(* CODESYS project Testment_Servo_Function_Test.export

Project tree, tasks and I/O mapping:
  Testment_Servo_Function_Test/
    program Servo_Testment_Main [ST]
    function block Testment_Message_Manager [ST]
*)

// Testment_Servo_Function_Test/Servo_Testment_Main
PROGRAM Servo_Testment_Main
VAR
	Set_Do: ARRAY [1..8] OF BOOL;
	Read_DI: ARRAY [1..12] OF BOOL;
	Read_DIA_Percentage :  ARRAY [0..7] OF REAL;
	Read_DIA_Raw :  ARRAY [0..7] OF UINT;
	
	// axis define
	FirstAxis : WORD := 1;
	LastAxis : WORD := 6;	// this value has been automaticlly asigned by global config reader
	//DI
	DI_Block : Digital_Input;
	
	//DO
	DO_Block : Digital_Output;
	
	//DIA
	smTime : TIME := T#250MS;
	DIA_Block : Digital_Input_Analog;
	
	
	// Testment functions
	Servo_Testment_State : INT := -1;
	Test_Process_Start_Restart, Error_State : BOOL;
	Message_Manager : Testment_Message_Manager;
	Show_Text : WSTRING;
	enb_axis : AuxAxis_PowerOn;
	read_axis : ARRAY [1..6] OF Arcalibrary.MCAT_ReadAxisMeasures;
	home_axis : ARRAY [1..6] OF Arcalibrary.MC_Home;
	re_j : INT;
	ts_i: INT;
	timer : ton;
	check_pos_err : REAL := 5;
	
	mov_axis : ARRAY [1..6] OF ArcaLibrary.MC_MoveAbsolute;
	FirstPos : REAL := 360;
	SecondPos : REAL := -360;
	CurrentPos : REAL;
	Vel : REAL := 180;
	Acc : REAL := 1900;
	Jerk : REAL := 9500;
	axis_mov_counter : INT;
	
	analog_cap ,analog_base : ARRAY [0..7] OF UINT;
	analog_difference : UINT := 12500; // 5v should be around 12900 ~ 13000
	set_override : ArcaLibrary.MC_GroupSetOverride;
	set_limit : ArcaLibrary.MCAT_AxisSetLimits;
	// analog control motor speed function
	analog_motor_state :INT := -1;
	debugButton : BOOL;
	speedLimit : REAL;
	analogFirPos : REAL := 380;
	analogSecPos : REAL := -380;
	analogVel : REAL := 18000;
	analogACC : REAL := 900000;
	analogJerk : REAL := 45000000;
	(* legacy ------
	forCounter: INT;
	//DI
	Read_6Ax_DI: Arcalibrary.ECAT_GetPdi_U32;
	DI_Raw : UDINT;
	new_DI_Value : UINT;
	
	//DO
	new_Do_Value, old_Do_Value : UINT;
	Write_6Ax_Do: Arcalibrary.ECAT_SetPdo_U32;
	------*)
	
	// servo elder program
	servo_elder_state :INT := -1;
	// elder_MoveType
	// 0 msans postion control all axis stop and turn in same time
	// 1 means speed control, two groups stop and turn in different times
	elder_MoveType : WORD := 1;
	elderVel : REAL := 18000;
	elderACC : REAL := 900000;
	elderJerk : REAL := 45000000;
	el_i : INT;
	speedFirGroup : ARRAY [0..5] OF ArcaLibrary.MC_MoveVelocity;
	speedSecGroup : ARRAY [0..5] OF ArcaLibrary.MC_MoveVelocity;
	elderTimer : ton;
	speedGroupSwitch : BOOL;
	speedSwitchTime : TIME := T#50MS;
	speedFirDir : ArcaLibrary.mc_Direction := mcPositiveDirection;
	speedSecDir : ArcaLibrary.mc_Direction := mcNegativeDirection;
	
	// 6 axis io test
	try: UINT;
	try2 : REAL;
	try3 : REAL := 3.9;
	read_0 : UINT;
	read_1 : UDINT;
	read_2 :ULINT;
	andValue : WORD;
	switch : BOOL;
	offsetValue : WORD := 147;
	TestAin_0: Arcalibrary.ECAT_GetPdi_U16;
	TestAin_1: Arcalibrary.ECAT_GetPdi_U32;
	TestAin_2: Arcalibrary.ECAT_GetPdi_U64;
	MaxmentOffset : UINT := 50;
	found_0, found_1, found_2, starter, maunl_next : BOOL;
	target_low : UINT := 12700;
	target_high : UINT := 13000;
	
	debugTimer : ton;
	FirstReachPos :  ARRAY [1..6] OF REAL := [0.6, -0.2, 0.606, -31.346, 178.434, 149.160];
	SecondReachPos :  ARRAY [1..6] OF REAL := [0.6, 0.2, 0.606, -31.346, 178.434, 149.160];
	Vell : REAL := 10;
	Accl : REAL := 10;
	Jerkl : REAL := 10;
	GrRelCorner :REAL := 0.5;
	MovErr : BOOL;
	//Movs : ARRAY [0..6] OF ArcaLibrary.MC_MoveLinearAbsolute;
	
	// error light control
	ErrLightControlState : INT;
	ErrLightTimer : Ton;
	ErrLightBlinkTime : TIME := T#200MS;
	ErrLightFinishTime : TIME := T#500MS;
	ErrLightCounterHigh : INT;
	ErrLightCounterLow : INT;
	ErrLight_i : INT;
	ErrLight_Switch : BOOL;
	// debug
	// --- because of homing bug (new servo need to home twice), get some function foe step 30
	homeErrOnce : BOOL;
	//---
	
	// debug
	manual_m01 : BOOL;
	manual_00 : BOOL;
	manual_20 : BOOL;
	manual_50 : BOOL;
	manual_jump_analog_check : BOOL;
	
	// debug para start---------------------------
	// read cfg message
	ReadCfg : ArcaLibrary.SYS_GetConfigInfo;
	Num_of_Axis:WORD;
	PowerState : ARRAY [0..5] OF ArcaLibrary.MCAT_ReadPowerStatus;
	AxisMeasure : ARRAY [0..5] OF ArcaLibrary.MCAT_ReadAxisMeasures;
	cfg_i : INT;
	
	//speed control test
	SC_Enb : BOOL; 
	SCMovTime : TIME := T#500MS;
	SCTimer : TON;
	SC_State : INT;
	SC_i,SC_y : INT;
	SpeedMovFir : ARRAY [0..5] OF ArcaLibrary.MC_MoveVelocity;
	SpeedMovSec : ARRAY [0..5] OF ArcaLibrary.MC_MoveVelocity;
	SCVel : REAL := 1800;
	SCACC : REAL := 9000;
	SCJerk : REAL := 45000;
	SCFirDir : ArcaLibrary.mc_Direction := mcPositiveDirection;
	SCSecDir : ArcaLibrary.mc_Direction := mcNegativeDirection;
	SCGroupSwitch : BOOL;
	
	// debug para end-----------------------------------
END_VAR

/////////////////////////////// instruction windows in chinsese  /////////////////////////////////////////

Message_Manager(state_in := Servo_Testment_State
	, start_restart_indicator => Test_Process_Start_Restart
	, Show_Message => Show_Text
	);
	
/////////////////////////////// instruction windows in chinsese  /////////////////////////////////////////

// if ethercat not ready then return
IF NOT ECatCfgok_GV THEN
	DI_Block (enable := FALSE);
	DO_Block (enable := FALSE);
	RETURN;
END_IF

IF Num_of_Axis_GV > 6 THEN
	Servo_Testment_State := -5;
END_IF
LastAxis := Num_of_Axis_GV;

DI_Block(enable := TRUE, DI_Array => Read_DI);
DO_Block(enable := TRUE, DO_Array := Set_Do);
DIA_Block(enable := TRUE, smoothTime := smTime
	, MaxRawInputValue := analog_cap
	, MinRawInputValue := analog_base
	, DIA_Raw => Read_DIA_Raw
	, DIA_Process => Read_DIA_Percentage
	);

enb_axis (enable := Servo_Testment_State > 9);
FOR re_j := 1 TO WORD_TO_INT(Num_of_Axis_GV) DO
	read_axis[re_j](axis := re_j - 1, enable :=  TRUE);
END_FOR

timer(in:= Servo_Testment_State = 30, pt := T#2S);

IF Servo_Testment_State <> -1 AND ((Read_DI[1] AND Read_DI[2]) OR manual_m01) THEN
	Servo_Testment_State := 0;
END_IF


set_limit(execute := debugButton, axis := 0, speedLimit := speedLimit); // useless

IF Servo_Testment_State < 130 THEN
	set_override(axesgroup := 0, enable := TRUE
	, velFactor := 1, accfactor := 1, jerkFactor := 1);
ELSE
	set_override(axesgroup := 0, enable := TRUE
	, velFactor := Read_DIA_Percentage[0]/100
	, accfactor := 1
	, jerkFactor := 1
	);
END_IF

IF Servo_Testment_State = 0 THEN	// reset
	//Set_Do[7]:= TRUE;
	//Set_Do[8]:= TRUE;
	homeErrOnce:= FALSE;
END_IF

CASE Servo_Testment_State OF
	-50: // analog cap and base difference too small
		// please connection and input voltage
		analog_cap[0];	// cap value
		analog_base[0];	// base vaule
	
	-45: // axis not mov to corrent pos
		ts_i; // error axis;
	-40: // if axis get err when moving
		ts_i; // error axis
	
	-35: // if some axis is not near 0 after homing
		ts_i; // error axis
		
	-33: // if some axis home err or time out
		ts_i;	// error axis
		
	-30: // if some axis home err
		home_axis[ts_i].ErrorID;	// homing err message
		
	-20: // if some axis can not enable
		enb_axis.Err_Message;	// enable err message
		
	-10: // if button is not commanding right inputs
		// plz check input button
		
	-5:	// config file contain more than 6 axis and exceed this program can handle
	
	-1:
		IF Read_DI[1] AND Read_DI[2] OR manual_m01 THEN
			Servo_Testment_State:= 0;
		ELSIF  Read_DI[1] OR Read_DI[2] THEN
			Servo_Testment_State := -10;	// if there is any input not receiving signal
		END_IF
		
	0:	// push second button to enable all axis
		IF Read_DI[3] AND Read_DI[4] AND Read_DI[5] AND Read_DI[6] OR manual_00 THEN
			Servo_Testment_State:= 10;
		ELSIF  Read_DI[3] OR Read_DI[4] OR Read_DI[5] OR Read_DI[6] THEN
			Servo_Testment_State := -10;	// if there is any input not receiving signal
		END_IF
	5:	// restart
		Servo_Testment_State := 10;
	10: // if 1~6 input is ok, waitting axis to enable
		IF enb_axis.Done THEN
			Servo_Testment_State := 20; // if enabled
		ELSIF enb_axis.Error THEN
			Servo_Testment_State := -20; // if some axis fail to enable
		END_IF
	20: // push third button to home axis
		FOR ts_i := WORD_TO_INT(FirstAxis) TO WORD_TO_INT(LastAxis) DO
			home_axis[ts_i](axis := ts_i - 1, execute := FALSE);	// reset blocks
		END_FOR
		IF Read_DI[7] AND Read_DI[8] AND Read_DI[9] OR homeErrOnce OR manual_20 THEN
			ts_i:= WORD_TO_INT(FirstAxis);
			Servo_Testment_State := 30;
		ELSIF Read_DI[7] OR Read_DI[8] OR Read_DI[9] THEN
			Servo_Testment_State := -10;	// if there is any input not receiving signal
		END_IF
	30: // start homing axis	// should not use I lkie in this case, is confilc with other state machine
		//Set_Do[7]:= TRUE;
		home_axis[ts_i](axis := ts_i - 1, execute := TRUE, position := 0, buffermode := mcAborting);
		IF home_axis[LastAxis].Done THEN	// all axis according to config file had homed
			FOR ts_i := WORD_TO_INT(FirstAxis) TO WORD_TO_INT(LastAxis) DO
				home_axis[ts_i](axis := ts_i - 1, execute := FALSE);
			END_FOR
			Servo_Testment_State := 40;
		ELSIF home_axis[ts_i].Done AND ts_i <= WORD_TO_INT(LastAxis) THEN // if current axis homing done
			timer(in:= FALSE);	// reset timer
			ts_i := ts_i + 1;
		ELSIF home_axis[ts_i].Error THEN	// if current axis get err
			Servo_Testment_State := -30;
		ELSIF timer.Q THEN	// if current axis not finish homing in certen time
			Servo_Testment_State := -33;
		END_IF
	40: // check if all axis are home
		ts_i := WORD_TO_INT(FirstAxis - 1);
		WHILE (ts_i < WORD_TO_INT(LastAxis)) AND Servo_Testment_State = 40 DO
			ts_i := ts_i + 1;
			IF read_axis[ts_i].Pos > check_pos_err OR read_axis[ts_i].Pos < -check_pos_err THEN // if current axis pos more than check_pos_err
				Servo_Testment_State := -35;
			END_IF
		END_WHILE
		IF Servo_Testment_State <> -35 THEN
			//Set_Do[8]:= TRUE;
			Servo_Testment_State := 50;
		END_IF
	50: // push fourth button to order motor turn
		FOR ts_i := WORD_TO_INT(FirstAxis) TO WORD_TO_INT(LastAxis) DO
			mov_axis[ts_i](axis := ts_i - 1, execute := FALSE);	// reset blocks
		END_FOR
		IF (Read_DI[10] AND Read_DI[11] AND Read_DI[12]) OR homeErrOnce OR manual_50 THEN
			Servo_Testment_State := 60;
		ELSIF Read_DI[10] OR Read_DI[11] OR Read_DI[12] THEN
			Servo_Testment_State := -10;	// if there is any input not receiving signal
		END_IF
	60:
		axis_mov_counter := 0;
		ts_i := WORD_TO_INT(FirstAxis - 1);
		WHILE ts_i < WORD_TO_INT(LastAxis) AND Servo_Testment_State = 60 DO
			ts_i := ts_i + 1;
			mov_axis[ts_i](axis := ts_i - 1, Execute := TRUE, Position := FirstPos
			, Velocity := vel, Acceleration := acc, Deceleration := Acc, jerk := jerk
			, Direction := mcShortestWay, BufferMode := mcAborting
			);
			IF mov_axis[ts_i].Done THEN
				axis_mov_counter := axis_mov_counter + 1;
			ELSIF  mov_axis[ts_i].Error THEN
				Servo_Testment_State := -40;	// axis err when moving
				IF NOT homeErrOnce THEN
					homeErrOnce := TRUE;
					Servo_Testment_State := 5;	// give secend chance
				END_IF
			END_IF
		END_WHILE
		IF axis_mov_counter >= WORD_TO_INT(LastAxis - (FirstAxis - 1)) AND Servo_Testment_State <> -40 THEN // if all axis mov done
			FOR ts_i := WORD_TO_INT(FirstAxis) TO WORD_TO_INT(LastAxis) DO
				mov_axis[ts_i](axis := ts_i - 1, execute := FALSE);	// reset blocks
			END_FOR
			Servo_Testment_State := 70;
		END_IF
	70: // check pos
		ts_i :=  WORD_TO_INT(FirstAxis - 1);
		WHILE ts_i < WORD_TO_INT(LastAxis) AND Servo_Testment_State = 70 DO
			ts_i := ts_i + 1;
			IF FirstPos - read_axis[ts_i].Pos < -check_pos_err OR FirstPos - read_axis[ts_i].Pos > check_pos_err THEN // if current axis pos more than check_pos_err
				Servo_Testment_State := -45;
			END_IF
		END_WHILE
		
		IF Servo_Testment_State <> -45 THEN
			Servo_Testment_State := 80;
		END_IF
		
	80: // motor start to turn
		axis_mov_counter := 0;
		ts_i := FirstAxis - 1;
		WHILE ts_i < WORD_TO_INT(LastAxis) AND Servo_Testment_State = 80 DO
			ts_i := ts_i + 1;
			mov_axis[ts_i](axis := ts_i - 1, Execute := TRUE, Position := SecondPos
			, Velocity := vel, Acceleration := acc, Deceleration := Acc, jerk := jerk
			, Direction := mcShortestWay, BufferMode := mcAborting
			);
			IF mov_axis[ts_i].Done THEN
				axis_mov_counter := axis_mov_counter + 1;
			ELSIF  mov_axis[ts_i].Error THEN
				Servo_Testment_State := -40;	// axis err when moving
			END_IF
		END_WHILE
		IF axis_mov_counter >= LastAxis - (FirstAxis - 1) AND Servo_Testment_State <> -40 THEN // if all axis mov done
			Servo_Testment_State := 90;
		END_IF
		
	90: // check pos
		ts_i := FirstAxis - 1;
		WHILE ts_i < WORD_TO_INT(LastAxis) AND Servo_Testment_State = 90 DO
			ts_i := ts_i + 1;
			IF SecondPos - read_axis[ts_i].Pos < -check_pos_err OR SecondPos - read_axis[ts_i].Pos > check_pos_err THEN // if current axis pos more than check_pos_err
				Servo_Testment_State := -45;
			END_IF
		END_WHILE
		IF Servo_Testment_State <> -45 THEN
			FOR ts_i := WORD_TO_INT(FirstAxis) TO WORD_TO_INT(LastAxis) DO
				mov_axis[ts_i](axis := ts_i - 1, execute := FALSE);	// reset blocks
			END_FOR
			Servo_Testment_State := 100;
		END_IF
		
	100: // set analog input base value, click second button to remember
		analog_base[0] := Read_DIA_Raw[0];
		IF Read_DI[3] AND Read_DI[4] AND Read_DI[5] AND Read_DI[6] OR manual_jump_analog_check THEN
			Servo_Testment_State:= 110;
		ELSIF  Read_DI[3] OR Read_DI[4] OR Read_DI[5] OR Read_DI[6] THEN
			Servo_Testment_State := -10;	// if there is any input not receiving signal
		END_IF
		
	110: // set analog input cap value, click third button to remember
		analog_cap[0] := Read_DIA_Raw[0];
		IF Read_DI[7] AND Read_DI[8] AND Read_DI[9] OR manual_jump_analog_check THEN
			Servo_Testment_State := 120;
		ELSIF Read_DI[7] OR Read_DI[8] OR Read_DI[9] THEN
			Servo_Testment_State := -10;	// if there is any input not receiving signal
		END_IF
		
	120: // check difference between cap and base
		IF (analog_cap[0] - analog_base[0] > analog_difference) OR manual_jump_analog_check THEN
			Servo_Testment_State := 130;
		ELSE
			Servo_Testment_State := -50;
		END_IF
	130:
		
	//100: // procedure done
		
END_CASE

(*IF Servo_Testment_State < 130 THEN
	analog_motor_state := -1;
END_IF

(*************
original Servo_Testment_State > 130 is designed for analog control axis speed
currently this state is use for servo elder testment
*******************)
CASE analog_motor_state	OF

	-1:
		//analog_motor_state := 0;
	0:
		FOR i := 1 TO WORD_TO_INT(Num_of_Axis_GV) DO	// should not use I here because this I is conflic with test state
			mov_axis[i](axis := i - 1, execute := FALSE);	// reset blocks
		END_FOR
		analog_motor_state := 10;
		debugTimer(in:= FALSE);
		(*
	10:
		mov_axis[1](axis := 0, Execute := TRUE, Position := 0);
		mov_axis[2](axis := 1, Execute := TRUE, Position := 0);
		mov_axis[3](axis := 2, Execute := TRUE, Position := 0);
		mov_axis[4](axis := 3, Execute := TRUE, Position := 0);
		mov_axis[5](axis := 4, Execute := TRUE, Position := 0);
		mov_axis[6](axis := 5, Execute := TRUE, Position := 0);
		debugTimer (in:= TRUE, pt := T#5S);
		IF debugTimer.Q THEN
			debugTimer(in:= FALSE);
			
			FOR i := 1 TO WORD_TO_INT(Num_of_Axis_GV) DO
				mov_axis[i](axis := i - 1, execute := FALSE);	// reset blocks
			END_FOR
			analog_motor_state := 20;
			
			Movs[0](axesgroup := 0, Execute := FALSE);
			
			Movs[1](axesgroup := 0, Execute := FALSE);
		END_IF
		
	20:
		Movs[0](axesgroup := 0, Execute := TRUE, Position := ADR(FirstReachPos)
			, Velocity := vell, Acceleration := accl, Deceleration := Accl, jerk := jerkl
			, coordsystem := mcMcs, BufferMode := mcAborting
			, TransitionMode := tmNone, TransitionParameter:=ADR(GrRelCorner)
			, Error => MovErr);
		IF Movs[0].Done THEN
			Movs[0](axesgroup := 0, Execute := FALSE);
			analog_motor_state := 30;
		END_IF
	30:
		Movs[1](axesgroup := 0, Execute := TRUE, Position := ADR(SecondReachPos)
			, Velocity := vell, Acceleration := accl, Deceleration := Accl, jerk := jerkl
			, coordsystem := mcMcs, BufferMode := mcAborting
			, TransitionMode := tmNone, TransitionParameter:=ADR(GrRelCorner)
			, Error => MovErr);
		IF Movs[1].Done THEN
			Movs[1](axesgroup := 0, Execute := FALSE);
			analog_motor_state := 20;
		END_IF
	*)
END_CASE*)

IF Servo_Testment_State < 130 THEN
	servo_elder_state := -1;
END_IF
CASE servo_elder_state OF
	-1:
		IF elder_MoveType = 0 THEN	// if control in abs 
			servo_elder_state := 0;
		ELSIF elder_MoveType = 1 THEN	// if control in vel
			servo_elder_state := 30;
		END_IF
	0:
		FOR el_i := 1 TO WORD_TO_INT(Num_of_Axis_GV) DO
			mov_axis[el_i](axis := el_i - 1, execute := FALSE);	// reset blocks
		END_FOR
		
		servo_elder_state := 10;
	10:
		axis_mov_counter := 0;
		el_i := 0;
		WHILE el_i < WORD_TO_INT(LastAxis - (FirstAxis - 1)) AND Servo_Testment_State <> -40 DO
			el_i := el_i + 1;
			mov_axis[el_i](axis := el_i - 1, Execute := TRUE, Position := analogFirPos
				, velocity := elderVel, Acceleration := elderACC, Deceleration := elderACC, Jerk := elderJerk
				, Direction := mcShortestWay, BufferMode := mcAborting
			);
			IF mov_axis[el_i].Done THEN
				axis_mov_counter := axis_mov_counter + 1;
			ELSIF  mov_axis[el_i].Error THEN
				Servo_Testment_State := -40;	// axis err when moving
			END_IF
		END_WHILE
		IF axis_mov_counter >= 6 AND Servo_Testment_State <> -40 THEN // if all axis mov done
			FOR el_i := WORD_TO_INT(FirstAxis) TO WORD_TO_INT(LastAxis) DO
				mov_axis[el_i](axis := el_i - 1, execute := FALSE);	// reset blocks
			END_FOR
			servo_elder_state := 20;
		END_IF
	20:
		axis_mov_counter := 0;
		el_i := 0;
		WHILE el_i < WORD_TO_INT(LastAxis - (FirstAxis - 1)) AND Servo_Testment_State <> -40 DO
			el_i := el_i + 1;
			mov_axis[el_i](axis := el_i - 1, Execute := TRUE, Position := analogSecPos
				, velocity := elderVel, Acceleration := elderACC, Deceleration := elderACC, Jerk := elderJerk
				, Direction := mcShortestWay, BufferMode := mcAborting
			);
			IF mov_axis[el_i].Done THEN
				axis_mov_counter := axis_mov_counter + 1;
			ELSIF  mov_axis[el_i].Error THEN
				Servo_Testment_State := -40;	// axis err when moving
			END_IF
		END_WHILE
		IF axis_mov_counter >= 6 AND Servo_Testment_State <> -40 THEN // if all axis mov done
			FOR el_i := WORD_TO_INT(FirstAxis) TO WORD_TO_INT(LastAxis) DO
				mov_axis[el_i](axis := el_i - 1, execute := FALSE);	// reset blocks
			END_FOR
			servo_elder_state := 10;
		END_IF
	30:
		FOR el_i := 0 TO 5 DO
			speedFirGroup[el_i](axis := el_i,execute := FALSE);
			speedSecGroup[el_i](axis := el_i,execute := FALSE);
		END_FOR
		elderTimer(in := FALSE);
		speedGroupSwitch := FALSE;
		servo_elder_state := 40;
	40:
		elderTimer(in := TRUE, pt := speedSwitchTime);
		IF elderTimer.Q THEN	// if time reached
			IF NOT speedGroupSwitch THEN	//decide which motor group is time to switch dir
				speedGroupSwitch := TRUE;
				IF speedFirDir = mcPositiveDirection THEN	// if first group is moving positivily
					speedFirDir := mcNegativeDirection;	// then switch to negative
				ELSE
					speedFirDir := mcPositiveDirection;
				END_IF
			ELSE
				speedGroupSwitch := FALSE;
				IF speedSecDir = mcPositiveDirection THEN
					speedSecDir := mcNegativeDirection;
				ELSE
					speedSecDir := mcPositiveDirection;
				END_IF
			END_IF
		END_IF
		FOR el_i := 0 TO 5 BY 2 DO
			speedFirGroup[el_i](axis := el_i,execute := NOT (elderTimer.Q AND speedGroupSwitch)	// only switch off when timer is alarted and first group direction is switched
				, velocity := elderVel, Acceleration := elderACC, Deceleration := elderACC, Jerk := elderJerk
				, Direction := speedFirDir, Buffermode := mcAborting);
			IF  speedFirGroup[el_i].Error THEN
				Servo_Testment_State := -40;	// axis err when moving
			END_IF
		END_FOR
		FOR el_i := 1 TO 5 BY 2 DO
			speedFirGroup[el_i](axis := el_i,execute := NOT (elderTimer.Q AND NOT speedGroupSwitch)	// only switch off when timer is alarted and second group direction is switched
				, velocity := elderVel, Acceleration := elderACC, Deceleration := elderACC, Jerk := elderJerk
				, Direction := speedSecDir, Buffermode := mcAborting);
			IF  speedFirGroup[el_i].Error THEN
				Servo_Testment_State := -40;	// axis err when moving
			END_IF
		END_FOR
		
		IF elderTimer.Q THEN	// if time reached
			elderTimer(in := FALSE);	// switch off timer
		END_IF
END_CASE

IF Servo_Testment_State > -1 THEN
	errlightcontrolstate := 0;
END_IF
CASE errlightcontrolstate OF
	0:
		Set_Do[7]:= TRUE;
		Set_Do[8]:= TRUE;
		IF Servo_Testment_State < 0 THEN
			Set_Do[7]:= FALSE;
			Set_Do[8]:= FALSE;
			ErrLightCounterHigh := (ABS(Servo_Testment_State) / 10) MOD 10;
			ErrLightCounterLow := ABS(Servo_Testment_State) MOD 10;
			ErrLightTimer(in := FALSE);
			ErrLight_i := 0;
			ErrLight_Switch := FALSE;
			IF ErrLightCounterHigh > 0 THEN
				errlightcontrolstate := 10;	// if there have higer num next state
			ELSE
				errlightcontrolstate := 20;	// go to low num directily
			END_IF
		END_IF
	10:	// blink higher number
		Set_Do[7]:= ErrLight_Switch;
		ErrLightTimer(in := TRUE , pt:= ErrLightBlinkTime);
		IF ErrLightTimer.Q THEN
			IF ErrLight_Switch THEN
				ErrLight_Switch := FALSE;
			ELSE
				ErrLight_Switch := TRUE;
			END_IF
			ErrLightTimer (in := FALSE);
			ErrLight_i := ErrLight_i + 1;
		END_IF
		IF ErrLight_i >= (ErrLightCounterHigh * 2) THEN
			ErrLightTimer(in := FALSE);
			ErrLight_i := 0;
			ErrLight_Switch := FALSE;
			IF ErrLightCounterLow > 0 THEN
				errlightcontrolstate := 20;	// if have lower num
			ELSE
				errlightcontrolstate := 30;	// go wating time
			END_IF
		END_IF
	20:// blink lower number
		Set_Do[8]:= ErrLight_Switch;
		ErrLightTimer(in := TRUE , pt:= ErrLightBlinkTime);
		IF ErrLightTimer.Q THEN
			IF ErrLight_Switch THEN
				ErrLight_Switch := FALSE;
			ELSE
				ErrLight_Switch := TRUE;
			END_IF
			ErrLightTimer (in := FALSE);
			ErrLight_i := ErrLight_i + 1;
		END_IF
		IF ErrLight_i >= (ErrLightCounterLow * 2) THEN
			ErrLightTimer(in := FALSE);
			ErrLight_i := 0;
			ErrLight_Switch := FALSE;
			errlightcontrolstate := 30;	// next state
		END_IF
	30:
		ErrLightTimer(in := TRUE, pt := ErrLightFinishTime);
		IF ErrLightTimer.Q THEN
			errlightcontrolstate := 0;
		END_IF
END_CASE

(* legacy ------
// read di
Read_6Ax_DI(Enable:=Num_of_axis_GV > 0, Offset:=143, Value=>DI_Raw);
new_DI_Value := UDINT_TO_UINT(DI_Raw);	// need convert to UINT otherwise it contain much more unwanted bits, it's not necessary but just keep this line to remember
// judge which bit is true
FOR forCounter := 1 TO UINT_TO_INT(SIZEOF(Read_DI)) DO // loop all bool value
	Read_DI[forCounter] := UINT_TO_BOOL(new_DI_Value AND SHL(1, forCounter - 1));
END_FOR

// write do
new_Do_Value:= 0;	// initialize 

(*	useless too complicated, no need to do the real calculation
FOR forCounter := 0 TO UINT_TO_INT(SIZEOF(SetDo)) DO // loop all bool value
	IF SetDo[forCounter] THEN	// if out put is true
		squareValue := 1;	// first value is 1, 2^0=1
		IF forCounter <> 0 THEN // if is not first value
			FOR squareCounter := 1 TO forCounter DO	// calculate dec value
				squareValue := squareValue * 2;
			END_FOR
		END_IF
		DoValue := DoValue + INT_TO_UINT(squareValue);
	END_IF
END_FOR
*)
// shift mamary according to bool
FOR forCounter := 1 TO UINT_TO_INT(SIZEOF(Set_Do)) DO // loop all bool value
	IF Set_Do[forCounter] THEN	// if out put is true
		new_Do_Value := new_Do_Value + SHL(1, forCounter - 1);
	END_IF
END_FOR

IF new_Do_Value <> old_Do_Value THEN
	old_Do_Value := new_Do_Value;
END_IF
Write_6Ax_Do(Enable:=Num_of_axis_GV > 0, Offset:=143, Value:=old_Do_Value);	// write DO
---------*)
// debug
IF NOT starter THEN
	starter := TRUE;
	found_0 := found_1 := found_2 := FALSE;
	offsetValue := 0;
END_IF
TestAin_0(enable:= TRUE, offset :=offsetValue, value=>read_0);
TestAin_1(enable:= TRUE, offset :=offsetValue, value=>read_1);
TestAin_2(enable:= TRUE, offset :=offsetValue, value=>read_2);

IF read_0 > try THEN
	try := read_0 - MaxmentOffset;
END_IF
try2 := (UINT_TO_REAL(read_0)/UINT_TO_REAL(try))*100;

IF read_0 > target_low AND read_0 < target_high THEN
	found_0 := TRUE;
END_IF

IF read_1 > target_low AND read_1 < target_high THEN
	found_1 := TRUE;
END_IF

IF read_2 > target_low AND read_2 < target_high THEN
	found_2 := TRUE;
END_IF

IF NOT found_0 AND NOT found_1 AND NOT found_2 OR maunl_next THEN
	offsetValue := offsetValue + 1;
	maunl_next := found_0 := found_1 := found_2 := FALSE;
END_IF

//Debug area start-------------------------------------------------------------------
// read how many axis has been config
ReadCfg(axisnumber => Num_of_axis);
FOR cfg_i := 0 TO WORD_TO_INT(Num_of_axis) - 1 DO
	PowerState[cfg_i](axis := cfg_i, enable := TRUE);
	AxisMeasure[cfg_i](axis := cfg_i, enable := TRUE);
	IF PowerState[cfg_i].State = 3 THEN // servo lost or error
		Servo_Testment_State := -40;
	END_IF
END_FOR


PowerState[0].State;
PowerState[1].State;
PowerState[2].State;
PowerState[3].State;
PowerState[4].State;
PowerState[5].State;
PowerState[0].Valid;
PowerState[1].Valid;
PowerState[2].Valid;
PowerState[3].Valid;
PowerState[4].Valid;
PowerState[5].Valid;
AxisMeasure[0].Valid;
AxisMeasure[1].Valid;
AxisMeasure[2].Valid;
AxisMeasure[3].Valid;
AxisMeasure[4].Valid;
AxisMeasure[5].Valid;
AxisMeasure[0].Pos;
AxisMeasure[1].Pos;
AxisMeasure[2].Pos;
AxisMeasure[3].Pos;
AxisMeasure[4].Pos;
AxisMeasure[5].Pos;
AxisMeasure[0].Speed;
AxisMeasure[1].Speed;
AxisMeasure[2].Speed;
AxisMeasure[3].Speed;
AxisMeasure[4].Speed;
AxisMeasure[5].Speed;
AxisMeasure[0].Torque;
AxisMeasure[1].Torque;
AxisMeasure[2].Torque;
AxisMeasure[3].Torque;
AxisMeasure[4].Torque;
AxisMeasure[5].Torque;
AxisMeasure[0].Acc;
AxisMeasure[1].Acc;
AxisMeasure[2].Acc;
AxisMeasure[3].Acc;
AxisMeasure[4].Acc;
AxisMeasure[5].Acc;

// speed control test
IF NOT sc_enb THEN
	SC_State := 0;
END_IF
CASE SC_State OF
	-10:	// error will moving
	0:
		IF SC_Enb THEN
			FOR sc_i := 0 TO 5 DO
				SpeedMovFir[sc_i](axis := sc_i,execute := FALSE);
				SpeedMovSec[sc_i](axis := sc_i,execute := FALSE);
			END_FOR
			SCTimer(in := FALSE);
			SCGroupSwitch := FALSE;
			sc_state := 10;
		END_IF
	10:
		SCTimer(in := TRUE, pt := SCMovTime);
		IF SCTimer.Q THEN	// if time reached
			IF NOT SCGroupSwitch THEN	//decide which motor group is time to switch dir
				SCGroupSwitch := TRUE;
				IF SCFirDir = mcPositiveDirection THEN	// if first group is moving positivily
					SCFirDir := mcNegativeDirection;	// then switch to negative
				ELSE
					SCFirDir := mcPositiveDirection;
				END_IF
			ELSE
				SCGroupSwitch := FALSE;
				IF SCSecDir = mcPositiveDirection THEN
					SCSecDir := mcNegativeDirection;
				ELSE
					SCSecDir := mcPositiveDirection;
				END_IF
			END_IF
		END_IF
		FOR sc_i := 0 TO 5 BY 2 DO
			SpeedMovFir[sc_i](axis := sc_i,execute := NOT (SCTimer.Q AND SCGroupSwitch)	// only switch off when timer is alarted and first group direction is switched
				, velocity := SCVel, Acceleration := SCACC, Deceleration := SCACC, Jerk := SCJerk
				, Direction := SCFirDir, Buffermode := mcAborting);
			IF SpeedMovFir[sc_i].Error THEN
				SC_State := -10;
			END_IF
		END_FOR
		FOR sc_i := 1 TO 5 BY 2 DO
			SpeedMovSec[sc_i](axis := sc_i,execute := NOT (SCTimer.Q AND NOT SCGroupSwitch)	// only switch off when timer is alarted and second group direction is switched
				, velocity := SCVel, Acceleration := SCACC, Deceleration := SCACC, Jerk := SCJerk
				, Direction := SCSecDir, Buffermode := mcAborting);
			IF SpeedMovSec[sc_i].Error THEN
				SC_State := -10;
			END_IF
		END_FOR
		
		IF SCTimer.Q THEN	// if time reached
			SCTimer(in := FALSE);	// switch off timer
		END_IF
END_CASE


//Debug area end-------------------------------------------------------------------

END_PROGRAM

// Testment_Servo_Function_Test/Testment_Message_Manager
FUNCTION_BLOCK Testment_Message_Manager
VAR_INPUT
	state_in : INT;
END_VAR
VAR_OUTPUT
	Start_Restart_indicator : BOOL;
	Show_Message : WSTRING;
	Error_State : BOOL;
END_VAR
VAR
	_case : int;
END_VAR

_case := state_in;

IF state_in < 0 THEN
	Error_State := TRUE;
ELSE 
	Error_State := FALSE;
END_IF

IF state_in <> 0 THEN
	Start_Restart_indicator := FALSE;
END_IF

CASE _case OF 
	-50:
		Show_Message := " 错误_50 ";
	-45:
		Show_Message := " 错误_45 ";
	-40:
		Show_Message := " 错误_40 ";
	-35:
		Show_Message := " 错误_35 ";
	-33:
		Show_Message := " 错误_33 ";
	-30:
		Show_Message := " 错误_30 ";
	-20:
		Show_Message := " 错误_20 ";
	-10:
		Show_Message := " 错误_10 ";
	-5:
		Show_Message := " 错误_5 ";
	0:
		Start_Restart_indicator := TRUE;
		Show_Message := " 步骤_0 ";
	20:
		Show_Message := " 步骤_20 ";
	50:
		Show_Message := " 步骤_50 ";
	100:
		Show_Message := " 步骤_100 ";
	110:
		Show_Message := " 步骤_110 ";
	130:
		Show_Message := " 步骤_130 ";
	
	//140:	
	//	Show_Message := " 完成 ";
	
END_CASE

END_FUNCTION_BLOCK
